# EPICS autosave request: iocBoot/ioc13test/auto_settings.req
file "sseq_settings.req",         P=$(P), S=SSEQ1
